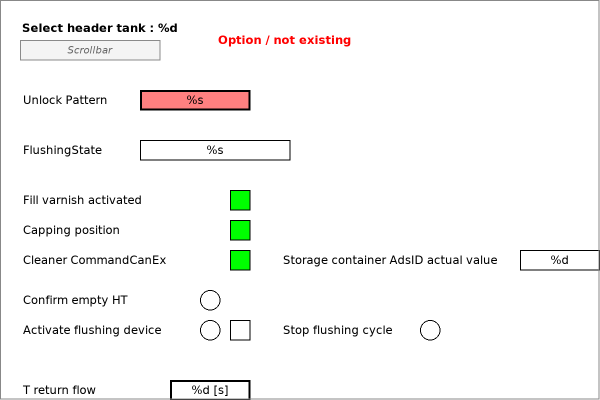
VISUALIZATION VISU_HT_FLUSHING_DEVICE  // 600x400
    Rectangle (20,190 160x20), "Fill varnish activated", invisible if: NOT PRG_INK.bL_FlushingUnlock
    Scrollbar (20,40 140x20), input disabled if: PRG_INK.bL_FlushingActive
        p2245068023: CONFIGURATION.iCIk_NB_HEADERTANK
        p1057716461: PRG_INK.iL_SelHeaderTankFlushing
    Rectangle (15,18 180x20), "Select header tank : %d", text variable: PRG_INK.iL_SelHeaderTankFlushing
    Rectangle (215,30 150x20), "Option / not existing", invisible if: bCIk_HEADERTANK_EXIST[PRG_INK.iL_SelHeaderTankFlushing]
    Rectangle (20,90 100x20), "Unlock Pattern"
    Rectangle (20,290 160x20), "Confirm empty HT", invisible if: NOT PRG_INK.bL_FlushingUnlock
    Rectangle (20,320 160x20), "Activate flushing device", invisible if: NOT PRG_INK.bL_FlushingUnlock
    Rectangle (20,380 110x20), "T return flow", invisible if: NOT PRG_INK.bL_FlushingUnlock
    Ellipse (200,320 20x20), colour toggle: PRG_INK.bL_FlushingActivate, invisible if: NOT PRG_INK.bL_FlushingUnlock
        toggle PRG_INK.bL_FlushingActivate
    RoundedRectangle (230,320 20x20), colour toggle: PRG_INK.bL_FlushingActive, invisible if: NOT PRG_INK.bL_FlushingUnlock
    Ellipse (200,290 20x20), colour toggle: PRG_INK.bL_FlushingHtEmpty, invisible if: NOT PRG_INK.bL_FlushingUnlock, input disabled if: NOT PRG_INK.bIKn_TankInkLevelReached[PRG_INK.iL_SelHeaderTankFlushing] OR PRG_INK.bL_FlushingActive
        toggle PRG_INK.bL_FlushingHtEmpty
    RoundedRectangle (230,190 20x20), colour toggle: PRG_INK.sAdsIkHeaderTank[PRG_INK.iL_SelHeaderTankFlushing].bI_EnableFillInk, invisible if: NOT PRG_INK.bL_FlushingUnlock
    Rectangle (170,380 80x20), "%d [s]", text variable: PRG_INK.lL_TimeFlushingReturnFlow, invisible if: NOT PRG_INK.bL_FlushingUnlock
        OnMouseDown: write the text variable via Edit
    Rectangle (140,90 110x20), "%s", text variable: PRG_INK.aI_FlushingSafePattern, colour toggle: PRG_INK.bL_FlushingUnlock
        OnMouseDown: write the text variable via Edit
    Rectangle (20,140 110x20), "FlushingState"
    Rectangle (140,140 150x20), "%s", text variable: PRG_INK.aL_FlushingState
    Rectangle (20,220 160x20), "Capping position", invisible if: NOT PRG_INK.bL_FlushingUnlock
    RoundedRectangle (230,220 20x20), colour toggle: NOT PRG_INK.bL_InCappingPos, invisible if: NOT PRG_INK.bL_FlushingUnlock
    Rectangle (280,320 130x20), "Stop flushing cycle", invisible if: NOT PRG_INK.bL_FlushingUnlock
    Ellipse (420,320 20x20), colour toggle: PRG_INK.bL_FlushingStop, invisible if: NOT PRG_INK.bL_FlushingUnlock
        toggle PRG_INK.bL_FlushingStop
    Rectangle (520,250 80x20), "%d", text variable: PRG_INK.sAdsIkHeaderTank[PRG_INK.iL_SelHeaderTankFlushing].sO_ActStoragetankAssignment.lI_Val, invisible if: NOT PRG_INK.bL_FlushingUnlock
        OnMouseDown: write the text variable via Edit
    Rectangle (280,250 230x20), "Storage container AdsID actual value", invisible if: NOT PRG_INK.bL_FlushingUnlock
    Rectangle (20,250 160x20), "Cleaner CommandCanEx", invisible if: NOT PRG_INK.bL_FlushingUnlock
    RoundedRectangle (230,250 20x20), colour toggle: NOT PRG_INK.sAdsIkHeaderTank[PRG_INK.iL_SelHeaderTankFlushing].sI_ActivateCleaner.bO_CommandCanEx, invisible if: NOT PRG_INK.bL_FlushingUnlock
END_VISUALIZATION

(* stored: Version 1.1.0.1, ProductVersion 3.1.4024.9
   Visu VISU_HT_FLUSHING_DEVICE: Id {f76c96d0-1438-44f8-98a0-996e33896124} *)
